FUNCTION_BLOCK FB_MotionAxisDS402 IMPLEMENTS I_MotionAxis
VAR_INPUT
END_VAR
VAR_OUTPUT
END_VAR
VAR
        AxisRef : REFERENCE TO AXIS_REF;
END_VAR

{warning 'Add method implementation '}
METHOD CalibrateEncValue
END_METHOD

{warning 'Add method implementation '}
METHOD EncSaveRestore
END_METHOD

{warning 'Add property implementation'}
PROPERTY Error : BOOL
GET
END_GET
END_PROPERTY

{warning 'Add property implementation'}
PROPERTY ErrorID : BOOL
GET
END_GET
END_PROPERTY

//FB_Init is always available implicitly and it is used primarily for initialization.
//The return value is not evaluated. For a specific influence, you can also declare the
//methods explicitly and provide additional code there with the standard initialization
//code. You can evaluate the return value.
METHOD FB_Init: BOOL
VAR_INPUT
    bInitRetains: BOOL; // TRUE: the retain variables are initialized (reset warm / reset cold)
    bInCopyCode: BOOL;  // TRUE: the instance will be copied to the copy code afterward (online change)
    AxisReference : REFERENCE TO AXIS_REF;
END_VAR
AxisRef REF= AxisReference;
END_METHOD

{warning 'Add method implementation '}
METHOD GearIn
END_METHOD

{warning 'Add method implementation '}
METHOD GearOut
END_METHOD

{warning 'Add method implementation '}
METHOD GetAxisRef : REFERENCE TO AXIS_REF
END_METHOD

{warning 'Add method implementation '}
METHOD GetPowerOverride : LREAL
END_METHOD

{warning 'Add method implementation '}
METHOD Halt
VAR_INPUT
    Deceleration	: LREAL := 0.0;
    Jerk	: LREAL := 0.0;
    BufferMode	: MC_BufferMode := .MC_BufferMode.MC_Aborting;
END_VAR
VAR_OUTPUT
    Done	: BOOL;
    Busy	: BOOL;
    Active	: BOOL;
    CommandAborted	: BOOL;
    Error	: BOOL;
    ErrorID	: UDINT;
    ErrorStr	: T_MaxString;
END_VAR
END_METHOD

{warning 'Add property implementation'}
PROPERTY HaltBusy : BOOL
GET
END_GET
END_PROPERTY

{warning 'Add property implementation'}
PROPERTY HaltDone : BOOL
GET
END_GET
END_PROPERTY

{warning 'Add property implementation'}
PROPERTY HaltError : BOOL
GET
END_GET
END_PROPERTY

{warning 'Add property implementation'}
PROPERTY HaltErrorID : UDINT
GET
END_GET
END_PROPERTY


METHOD Home
VAR_INPUT
    Position : LREAL := DEFAULT_HOME_POSITION;
    HomingMode : MC_HomingMode := MC_DefaultHoming;
END_VAR
VAR_OUTPUT
    Done	: BOOL;
    Busy	: BOOL;
    Active	: BOOL;
    CommandAborted	: BOOL;
    Error	: BOOL;
    ErrorID	: UDINT;
    ErrorStr	: T_MaxString;
END_VAR
END_METHOD

{warning 'Add property implementation'}
PROPERTY HomeBusy : BOOL
GET
END_GET
END_PROPERTY

{warning 'Add property implementation'}
PROPERTY HomeDone : BOOL
GET
END_GET
END_PROPERTY

{warning 'Add property implementation'}
PROPERTY MeasuredAcceleration : LREAL
GET
END_GET
END_PROPERTY

{warning 'Add property implementation'}
PROPERTY MeasuredPosition : LREAL
GET
END_GET
END_PROPERTY

{warning 'Add property implementation'}
PROPERTY MeasuredVelocity : LREAL
GET
END_GET
END_PROPERTY

{warning 'Add method implementation '}
METHOD MoveAbsolute
VAR_INPUT
    Position	: LREAL;
    Velocity	: LREAL;
    Acceleration	: LREAL := 0.0;
    Deceleration	: LREAL := 0.0;
    Jerk	: LREAL := 0.0;
    BufferMode	: MC_BufferMode := .MC_BufferMode.MC_Aborting;
END_VAR
VAR_OUTPUT
    Done	: BOOL;
    Busy	: BOOL;
    Active	: BOOL;
    CommandAborted	: BOOL;
    Error	: BOOL;
    ErrorID	: UDINT;
    ErrorStr	: T_MaxString;
END_VAR
END_METHOD

{warning 'Add property implementation'}
PROPERTY MoveAbsoluteBusy : BOOL
GET
END_GET
END_PROPERTY

{warning 'Add property implementation'}
PROPERTY MoveAbsoluteDone : BOOL
GET
END_GET
END_PROPERTY

{warning 'Add property implementation'}
PROPERTY MoveAbsoluteError : BOOL
GET
END_GET
END_PROPERTY

{warning 'Add property implementation'}
PROPERTY MoveAbsoluteErrorID : UDINT
GET
END_GET
END_PROPERTY

{warning 'Add property implementation'}
PROPERTY MoveAbsoluteTargetAcceleration : LREAL
GET
END_GET
END_PROPERTY

{warning 'Add property implementation'}
PROPERTY MoveAbsoluteTargetDeceleration : LREAL
GET
END_GET
END_PROPERTY

{warning 'Add property implementation'}
PROPERTY MoveAbsoluteTargetJerk : LREAL
GET
END_GET
END_PROPERTY

{warning 'Add property implementation'}
PROPERTY MoveAbsoluteTargetPosition : LREAL
GET
END_GET
END_PROPERTY

{warning 'Add property implementation'}
PROPERTY MoveAbsoluteTargetVelocity : LREAL
GET
END_GET
END_PROPERTY

{warning 'Add property implementation'}
PROPERTY MoveBusy : BOOL
GET
END_GET
END_PROPERTY

{warning 'Add property implementation'}
PROPERTY MoveDone : BOOL
GET
END_GET
END_PROPERTY

{warning 'Add property implementation'}
PROPERTY NegativeMotionIsEnabled : BOOL
GET
END_GET
END_PROPERTY

{warning 'Add property implementation'}
PROPERTY PositiveMotionIsEnabled : BOOL
GET
END_GET
END_PROPERTY

{warning 'Add method implementation '}
METHOD Power
VAR_INPUT
    Enable	: BOOL;
    Enable_Positive	: BOOL;
    Enable_Negative	: BOOL;
    (* in percent from 0 to 100 *)
    Override	: LREAL := 100.0;
    BufferMode	: MC_BufferMode := .MC_BufferMode.MC_Aborting;
END_VAR
VAR_OUTPUT
    Status	: BOOL;
    Busy	: BOOL;
    Active	: BOOL;
    Error	: BOOL;
    ErrorID	: UDINT;
    ErrorStr	: T_MaxString;
END_VAR
END_METHOD

{warning 'Add property implementation'}
PROPERTY PowerError : BOOL
GET
END_GET
END_PROPERTY

{warning 'Add property implementation'}
PROPERTY PowerErrorID : UDINT
GET
END_GET
END_PROPERTY

{warning 'Add property implementation'}
PROPERTY PowerIsEnabled : BOOL
GET
END_GET
END_PROPERTY

{warning 'Add property implementation'}
PROPERTY PowerOverride : LREAL
GET
END_GET
END_PROPERTY

{warning 'Add property implementation'}
PROPERTY PowerStatus : BOOL
GET
END_GET
END_PROPERTY

{warning 'Add method implementation '}
METHOD Reset
VAR_OUTPUT
    Done	: BOOL;
    Busy	: BOOL;
    Error	: BOOL;
    ErrorID	: UDINT;
    ErrorStr	: T_MaxString;
END_VAR
END_METHOD

{warning 'Add property implementation'}
PROPERTY ResetBusy : BOOL
GET
END_GET
END_PROPERTY

{warning 'Add property implementation'}
PROPERTY ResetDone : BOOL
GET
END_GET
END_PROPERTY

{warning 'Add property implementation'}
PROPERTY ResetError : BOOL
GET
END_GET
END_PROPERTY

{warning 'Add property implementation'}
PROPERTY ResetErrorID : UDINT
GET
END_GET
END_PROPERTY

{warning 'Add property implementation'}
PROPERTY SetpointAcceleration : LREAL
GET
END_GET
END_PROPERTY

{warning 'Add property implementation'}
PROPERTY SetpointJerk : LREAL
GET
END_GET
END_PROPERTY

{warning 'Add property implementation'}
PROPERTY SetpointPosition : LREAL
GET
END_GET
END_PROPERTY

{warning 'Add property implementation'}
PROPERTY SetpointVelocity : LREAL
GET
END_GET
END_PROPERTY

{warning 'Add method implementation '}
METHOD SetPowerOverride
VAR_INPUT
    (* in percent from 0 to 100 *)
    Override	: LREAL;
END_VAR
VAR_OUTPUT
    Status	: BOOL;
    Busy	: BOOL;
    Active	: BOOL;
    Error	: BOOL;
    ErrorID	: UDINT;
    ErrorStr	: T_MaxString;
END_VAR
END_METHOD

END_FUNCTION_BLOCK

(* stored: Version 1.1.0.1
   POU FB_MotionAxisDS402: Id {e6939303-1a29-4526-8cba-ad7b7e0a797c}, SpecialFunc None
   Method CalibrateEncValue: Id {c7dcbcfa-a780-4c13-83ee-dd3a3259e8a3}
   Method EncSaveRestore: Id {758fc86b-abf1-47a5-8f0f-d4ef3c0ab63d}
   Property Error: Id {cac518e7-c4c8-4f02-a58c-d3e7d2d79cd8}
   Get Get: Id {1f4a15a1-4924-401f-9889-63882261a5e7}
   Property ErrorID: Id {0921f86d-40cd-4df8-ab28-2898c44fa05e}
   Get Get: Id {8966b06b-b307-481c-b0a4-39b5860997da}
   Method FB_Init: Id {180fa942-a7f1-463e-8d13-f7f31c42583f}
   Method GearIn: Id {bd71ffe0-808b-46c3-b7c4-4726451849e9}
   Method GearOut: Id {2f2fbcf8-48b9-4907-94c3-c4b4bd82d7a2}
   Method GetAxisRef: Id {70970299-6294-431d-9776-54d7232b96ee}
   Method GetPowerOverride: Id {49fbbd23-2407-4a66-ae5b-2e18cb4981be}
   Method Halt: Id {0d0d9db3-d251-4c98-9ee5-9c7cabbfae92}
   Property HaltBusy: Id {d5f36f64-1a55-4d41-a9c2-c76317220329}
   Get Get: Id {42083908-85a4-4f3d-92af-233c0686bc20}
   Property HaltDone: Id {d9c4a5e0-2ab3-40f5-9994-0eb6f9d01433}
   Get Get: Id {d16c9e22-5d30-483a-b808-c9aae656db15}
   Property HaltError: Id {5cfd0afa-c6b4-4b7b-b1d8-bb124ec37fdc}
   Get Get: Id {25e8bafc-b207-40a1-a2ef-9cefff41729c}
   Property HaltErrorID: Id {786f40cf-1067-458f-98f2-6541393330db}
   Get Get: Id {3b06a852-b6f5-475c-9fc8-4862cb335a53}
   Method Home: Id {c1e21c0a-478a-4e64-ac1c-4da91135d244}
   Property HomeBusy: Id {0b614afd-f884-405d-a3c9-940069cf0094}
   Get Get: Id {223b0e5f-eb6e-47c2-a3c7-5787f373de75}
   Property HomeDone: Id {71a6249c-03b6-4d17-9f52-bb3ed3787205}
   Get Get: Id {ad2908a1-2ddd-4a33-9355-57e43968bd13}
   Property MeasuredAcceleration: Id {934d9697-a40f-4eb9-a7f7-67ee6985cc2f}
   Get Get: Id {e0ab7cc1-6634-4353-9667-b1c724ec3f2d}
   Property MeasuredPosition: Id {2a84fca6-0f9b-4280-b2ca-2049fcfb94bd}
   Get Get: Id {a6a4bb59-026a-4928-9c9b-df4598680652}
   Property MeasuredVelocity: Id {efb2b425-b568-4bdf-833b-5bc65db366a5}
   Get Get: Id {cda91a7e-e3af-4435-9ed1-45de112df9a3}
   Method MoveAbsolute: Id {b79a8962-0b6c-4e26-8a83-40993f407295}
   Property MoveAbsoluteBusy: Id {0790109c-56c3-4e19-b6c2-acb92c392cb4}
   Get Get: Id {3d201901-9a75-4553-a5fa-ff6fe54d4d7a}
   Property MoveAbsoluteDone: Id {faeaacd2-8a9d-415c-9a78-e670be07b3d2}
   Get Get: Id {7f54dfdf-b07b-43f6-a310-d8d65b8720b6}
   Property MoveAbsoluteError: Id {4e493c61-094a-4389-995a-30e3946962cd}
   Get Get: Id {ed3b3d18-5d2e-4637-86ea-b9254eb9d0c5}
   Property MoveAbsoluteErrorID: Id {17e71446-17ad-4326-9132-290dafd4cf95}
   Get Get: Id {5ef70246-ab88-49b6-9f00-b8346a776b02}
   Property MoveAbsoluteTargetAcceleration: Id {642747c5-2103-4fe7-a4be-f191a1d64a90}
   Get Get: Id {cc1dfd9e-5ea9-416b-ab11-d1f7798db597}
   Property MoveAbsoluteTargetDeceleration: Id {e3db52ec-2501-41b8-b3ec-7be41fd21e1b}
   Get Get: Id {5eda09d2-41e2-4a9e-90b3-b7124ee9a43a}
   Property MoveAbsoluteTargetJerk: Id {70798a58-70dc-4808-a405-d9ca44e190c1}
   Get Get: Id {686b5815-904d-4225-bc40-f7da9e53721d}
   Property MoveAbsoluteTargetPosition: Id {2c8be390-cc7e-4683-9c6c-e00b2832638d}
   Get Get: Id {634b2890-d916-4ecb-be59-0a3fd804b486}
   Property MoveAbsoluteTargetVelocity: Id {9aff5306-41b3-4638-9345-15453e87a59d}
   Get Get: Id {0f80d99b-6f11-4c05-a4ea-dea851e710c2}
   Property MoveBusy: Id {be5040ac-8ff2-4ec4-93df-83ebd8969c60}
   Get Get: Id {7ed734b0-29b8-442a-975e-fc096e88aa06}
   Property MoveDone: Id {51fa4c87-afdd-47a9-8ad1-66b50ff00d39}
   Get Get: Id {48eb093d-9bb9-4989-a9a6-52ae56edd306}
   Property NegativeMotionIsEnabled: Id {7436ed1f-8644-4767-a7b5-08e16f5bc0a0}
   Get Get: Id {82bdc18b-2a7d-4d47-9621-01a7daccf2f2}
   Property PositiveMotionIsEnabled: Id {138ca617-0311-48a2-b19f-9e05794a76aa}
   Get Get: Id {f8bacf70-521b-46ae-879e-223de80f5c38}
   Method Power: Id {19d5d4aa-b380-44c1-a057-53da5a253fbc}
   Property PowerError: Id {68e594af-d141-444e-90dd-82d59426c017}
   Get Get: Id {13ad7120-04ca-4246-8e27-b7d429f86465}
   Property PowerErrorID: Id {e51792b2-d6f8-4544-a4f6-a19a4ee87bed}
   Get Get: Id {7bf2a67f-e3f8-4a07-bc29-e7f263650237}
   Property PowerIsEnabled: Id {2378d27c-639d-4a59-acb6-f7785b054605}
   Get Get: Id {1c39cdf1-d58d-47fd-8958-e56759420fbf}
   Property PowerOverride: Id {276994d9-1b30-4079-a978-8003304548f3}
   Get Get: Id {899ce412-1fd3-4721-8996-5169d30d1796}
   Property PowerStatus: Id {7a605967-f92b-43b5-8bb0-9eb4ff790479}
   Get Get: Id {fb0c8156-d81b-4a08-982e-f83282b7374a}
   Method Reset: Id {3a445482-f12e-4a74-b8f7-8f9d0d15c6fe}
   Property ResetBusy: Id {015960b6-b417-4a95-91bc-e811cafb6fd2}
   Get Get: Id {f34af71f-c5e9-490e-ba86-31a741a78b9e}
   Property ResetDone: Id {d72edc02-6959-4ad1-a60d-5e7dceee9c41}
   Get Get: Id {879bcbb1-8340-4158-a03e-c7eff304f738}
   Property ResetError: Id {c5e41283-8bb8-4748-85d7-15fdf5f10da2}
   Get Get: Id {03f3b9f6-75f5-4240-ada3-32128b6ed529}
   Property ResetErrorID: Id {3a03d3ac-e2bf-4529-9ced-682e011838f7}
   Get Get: Id {2bca9035-764c-438e-a7fd-d11436e0bb6d}
   Property SetpointAcceleration: Id {2b173762-6328-4e4c-95a8-b0b12612577c}
   Get Get: Id {d5868310-b848-4212-9134-fbd16e577603}
   Property SetpointJerk: Id {cb34f141-25c4-4329-957c-2f43fad59182}
   Get Get: Id {d9db7ea2-f8ce-4019-8c3c-40fdaa823278}
   Property SetpointPosition: Id {646f602a-22b9-4e57-88d7-81645cf1ef98}
   Get Get: Id {c7b5ce4f-fd1c-4607-8ae3-2f7f9a9d315c}
   Property SetpointVelocity: Id {75af3429-3580-4fd1-aa71-20f5f83b23b6}
   Get Get: Id {f94d94cf-9d1a-440b-a311-94bd32652378}
   Method SetPowerOverride: Id {d2b8fabe-aac6-4f1a-a530-9a80a3f12907} *)
